FUNCTION TryConvert_DINT_TO_LINT : BOOL
VAR_INPUT
	in : DINT;
	out : REFERENCE TO LINT;
END_VAR

out := DINT_TO_LINT(in);
TryConvert_DINT_TO_LINT := TRUE;

END_FUNCTION

(* stored: Version 1.1.0.1, ProductVersion 3.1.4024.12
   POU TryConvert_DINT_TO_LINT: Id {5539e4cc-b68b-4d9e-a750-7992db076dbc}, SpecialFunc None *)
